// TIA Portal V20 export
DATA_BLOCK "SP203"   // DB346
// stored: MemoryReserve 100
   VAR
      "MAIN OP MODE SLELECT SS.AUTO" : Bool := FALSE;
      "MAIN OP HOME PBL (GREEN)" : Bool := FALSE;
      "MAIN OP SAFETY RESET PBL (BLUE)" : Bool := FALSE;
      "MAIN OP SCS MODE SLELECT SS.AUTO" : Bool := FALSE;
      "MAIN OP MODE SLELECT SS.MANUAL" : Bool := TRUE;
      "MAIN OP ENABLE PBL (WHITE)" : Bool := FALSE;
      "MAIN OP SCS MODE SLELECT SS.SETUP" : Bool := TRUE;
      "MAIN OP SCS MODE SLELECT SS.DISABLE" : Bool := FALSE;
   END_VAR
BEGIN
END_DATA_BLOCK
